TYPE ST_PROCESS_DATA :
STRUCT
  ActiveStations      : T_PROCESS; // where and how many stations are to be used in process
  ProcessTarget       : UINT;      // for whom?
END_STRUCT
END_TYPE

(* stored: Version 1.1.0.1, ProductVersion 3.1.4024.13
   DUT ST_PROCESS_DATA: Id {89d728c0-a3cf-4c7f-a1e5-ad3df6f9ba44} *)
